///EL1859 | HD EtherCAT Terminal, 8-channel digital input + 8-channel digital output 24 V DC
FUNCTION_BLOCK EL1859

VAR_INPUT
	En: BOOL;
	bDo_1: BOOL;
	bDo_2: BOOL;
	bDo_3: BOOL;
	bDo_4: BOOL;
	bDo_5: BOOL;
	bDo_6: BOOL;
	bDo_7: BOOL;
	bDo_8: BOOL;
	iTerminal_ID : INT;
	ErrorSystem : POINTER TO ST_ErrorSystem;
END_VAR

VAR_OUTPUT
	EnO: BOOL;
	bDi_1: BOOL;
	bDi_2: BOOL;
	bDi_3: BOOL;
	bDi_4: BOOL;
	bDi_5: BOOL;
	bDi_6: BOOL;
	bDi_7: BOOL;
	bDi_8: BOOL;
	bError: BOOL;
END_VAR

VAR
	Channel_1_Input AT %I*: BOOL;
	Channel_2_Input AT %I*: BOOL;
	Channel_3_Input AT %I*: BOOL;
	Channel_4_Input AT %I*: BOOL;
	Channel_5_Input AT %I*: BOOL;
	Channel_6_Input AT %I*: BOOL;
	Channel_7_Input AT %I*: BOOL;
	Channel_8_Input AT %I*: BOOL;
	Channel_1_Output AT %Q*: BOOL;
	Channel_2_Output AT %Q*: BOOL;
	Channel_3_Output AT %Q*: BOOL;
	Channel_4_Output AT %Q*: BOOL;
	Channel_5_Output AT %Q*: BOOL;
	Channel_6_Output AT %Q*: BOOL;
	Channel_7_Output AT %Q*: BOOL;
	Channel_8_Output AT %Q*: BOOL;
	WcState_WcState AT %I*: BOOL;
	InfoData_State AT %I*: UINT;
	
	//FB-s
	fbTerminalError : FB_TerminalError;
END_VAR

EnO:=En;

//Error FB instance
fbTerminalError(
	En := TRUE,
	iTerminal_ID := iTerminal_ID,
	bWcState := WcState_WcState,
	uiInfoData_State := InfoData_State,
	pErrorSystem := ErrorSystem,
	bError => bError,
);

IF En THEN
	IF bError=FALSE THEN
		bDi_1:=Channel_1_Input;
		bDi_2:=Channel_2_Input;
		bDi_3:=Channel_3_Input;
		bDi_4:=Channel_4_Input;
		bDi_5:=Channel_5_Input;
		bDi_6:=Channel_6_Input;
		bDi_7:=Channel_7_Input;
		bDi_8:=Channel_8_Input;
		Channel_1_Output:=bDo_1;
		Channel_2_Output:=bDo_2;
		Channel_3_Output:=bDo_3;
		Channel_4_Output:=bDo_4;
		Channel_5_Output:=bDo_5;
		Channel_6_Output:=bDo_6;
		Channel_7_Output:=bDo_7;
		Channel_8_Output:=bDo_8;
	ELSE
		bDi_1:=FALSE;
		bDi_2:=FALSE;
		bDi_3:=FALSE;
		bDi_4:=FALSE;
		bDi_5:=FALSE;
		bDi_6:=FALSE;
		bDi_7:=FALSE;
		bDi_8:=FALSE;
	END_IF
END_IF

END_FUNCTION_BLOCK

(* stored: Version 1.1.0.1, ProductVersion 3.1.4022.10
   POU EL1859: Id {64929902-5a7b-4bb2-95c1-e538c2dbc480}, SpecialFunc None *)
